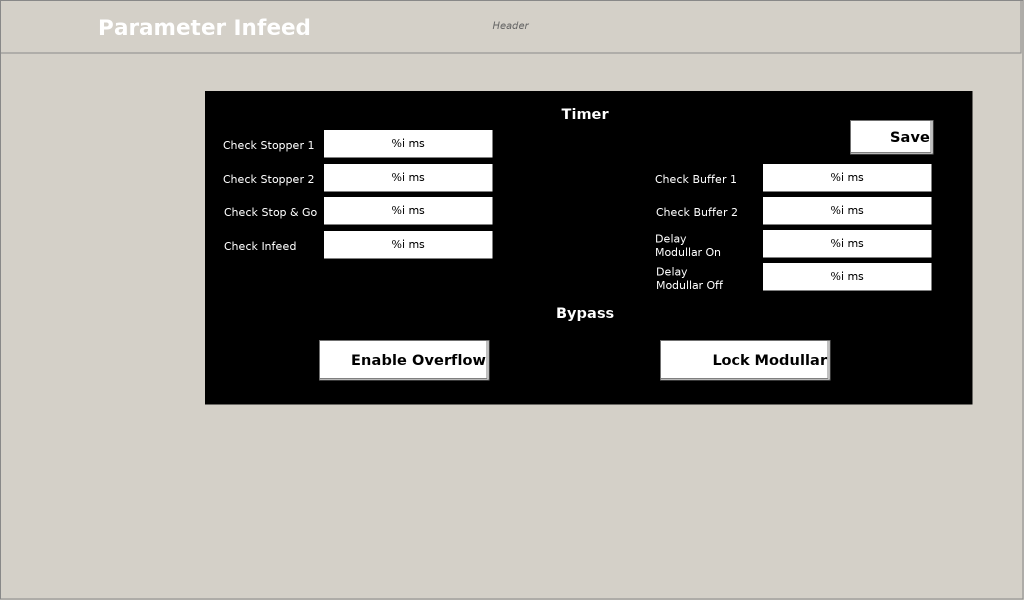
VISUALIZATION MInfeed  // 1024x600
    Frame (0,-2 1021x55)
        shows Header()
    Label (95,15 250x25), "Parameter Infeed"
    RoundedRectangle (205,91 767x313)
    Label (233,94 704x40), "Timer"
    Label (220,128 103x35), "Check Stopper 1"
    RoundedRectangle (323,129 170x29), "%i ms", text variable: HMI_GVL.Tmr_Stopper1
        OnMouseClick: write the text variable via Default
    Button (850,120 83x34), "Save", image: VisuSymbols.Symbols.Save
        tap InputOutput_GVL.TestMode[100]
    Label (220,162 104x35), "Check Stopper 2"
    RoundedRectangle (323,163 170x29), "%i ms", text variable: HMI_GVL.Tmr_Stopper2
        OnMouseClick: write the text variable via Default
    Label (652,162 102x35), "Check Buffer 1"
    RoundedRectangle (762,163 170x29), "%i ms", text variable: HMI_GVL.Tmr_Buffer1
        OnMouseClick: write the text variable via Default
    Label (221,195 102x35), "Check Stop & Go"
    RoundedRectangle (323,196 170x29), "%i ms", text variable: HMI_GVL.Tmr_StopGo
        OnMouseClick: write the text variable via Default
    Label (653,195 102x35), "Check Buffer 2"
    RoundedRectangle (762,196 170x29), "%i ms", text variable: HMI_GVL.Tmr_Buffer2
        OnMouseClick: write the text variable via Default
    Label (221,229 100x35), "Check Infeed"
    RoundedRectangle (323,230 170x29), "%i ms", text variable: HMI_GVL.Tmr_Infeed
        OnMouseClick: write the text variable via Default
    Label (233,293 704x40), "Bypass"
    Button (660,340 170x40), "Lock Modullar", colour toggle: HMI_GVL.LockModullarToRun, image: VisuSymbols.Symbols.Lock
        toggle HMI_GVL.LockModullarToRun
    Label (652,228 102x35), "Delay Modullar On"
    RoundedRectangle (762,229 170x29), "%i ms", text variable: HMI_GVL.Tmr_ModullarOn
        OnMouseClick: write the text variable via Default
    Label (653,261 102x35), "Delay Modullar Off"
    RoundedRectangle (762,262 170x29), "%i ms", text variable: HMI_GVL.Tmr_ModullarOff
        OnMouseClick: write the text variable via Default
    Button (319,340 170x40), "Enable Overflow", colour toggle: HMI_GVL.Disable_Overflow, image: VisuSymbols.Symbols.Lock
        toggle HMI_GVL.Disable_Overflow
END_VISUALIZATION

(* stored: Version 1.1.0.1, ProductVersion 3.1.4024.12
   Visu MInfeed: Id {659f4e56-0057-4b01-9d18-dc2294a6578c} *)
